FUNCTION_BLOCK Component EXTENDS FB_ComponentBase
VAR
	ComponentAlarms	 : ARRAY[1..COMPONENT_ALARM_COUNT] OF FB_TcAlarm;
	testError		 : BOOL;
	_ErrorSeverity	 : INT := 2;
	_WarningSeverity : INT;
END_VAR

VAR CONSTANT
	COMPONENT_ALARM_COUNT : UDINT := 7; //First is InitReferenceEvent
END_VAR

METHOD ChangeAlarmSeverity
CASE _WarningSeverity OF
	0:
		_ParentFaultResponseDefinitions[TcEventSeverity.Warning] := E_AlarmResponse.NoResponse;

	1:
		_ParentFaultResponseDefinitions[TcEventSeverity.Warning] := E_AlarmResponse.Abort_Immediate;

	2:
		_ParentFaultResponseDefinitions[TcEventSeverity.Warning] := E_AlarmResponse.Abort_ImmediateError;
END_CASE

CASE _ErrorSeverity OF
	0:
		_ParentFaultResponseDefinitions[TcEventSeverity.Error] := E_AlarmResponse.NoResponse;

	1:
		_ParentFaultResponseDefinitions[TcEventSeverity.Error] := E_AlarmResponse.Abort_Immediate;

	2:
		_ParentFaultResponseDefinitions[TcEventSeverity.Error] := E_AlarmResponse.Abort_ImmediateError;
END_CASE
END_METHOD

// Initializes event function blocks using this components's name
METHOD PROTECTED CreateEvents

// This method is called by Initialize() as required
F_CreateAllEventsInClass(Alarms		:= ComponentAlarms,
						 ClassSize	:= SIZEOF(TC_Events.Events_Component),
						 pInitEvent := ADR(TC_EVENTS.Events_Component.InitReferenceEvent),
						 Prefix		:= Name);

SUPER^.CreateEvents();
END_METHOD

// This method serves as the entry point for all underlying FB logic
METHOD PUBLIC CyclicLogic

// This method should be called cyclically by descendant function blocks by invoking SUPER^.CyclicLogic().  Alternatively, the contents of this method could be reimplemented entirely in which case a call to this method would not be necessary.
IF NOT _InitComplete THEN
	_InitComplete := Initialize();
	RETURN;
END_IF

//
ChangeAlarmSeverity();
SUPER^.CyclicLogic();

(*
*
*		Code must be after SUPER^.CyclicLogic();
*
*)

// Update alarm severity for this component
_CurrentAlarmSeverity := F_GetMaxSeverityRaised(Alarms := ComponentAlarms, CurrentSeverity := _CurrentAlarmSeverity);
_Error				  := _CurrentAlarmSeverity >= TcEventSeverity.Error;
END_METHOD

// Provides basic error detection and event handling for this component
METHOD PROTECTED Monitoring

//This method is called cyclically by CyclicLogic()
_Busy := FALSE;

//AlarmMonitoring
IF testError AND NOT ComponentAlarms[E_Events_Component.Error].bRaised THEN
	RaiseAlarm2Args(ComponentAlarms[E_Events_Component.Error], 'Note 1', 'Note 2');
END_IF

SUPER^.Monitoring();
END_METHOD

METHOD RaiseAlarm2Args
VAR_IN_OUT
	Alarm : FB_TcAlarm; //Alarm to be raised
END_VAR

VAR_INPUT
	String_1 : STRING; //First String Parameter (The Name of this component will be applied first automatically)
	String_2 : STRING; //Second String Parameter
END_VAR
F_RaiseAlarmWithStringParameters(Alarm	  := Alarm,
								 String_1 := Name,
								 String_2 := String_1,
								 String_3 := String_2);
END_METHOD

// Clears error flags and error IDs for this component
METHOD PUBLIC Reset : BOOL

//Typically called by the EMs SUPER^.Clearing Method
F_ClearAllEventsInClass(Alarms := ComponentAlarms);
IF SUPER^.Reset() THEN
	_Error	 := FALSE;
	_ErrorID := 0;
	Reset	 := TRUE;
END_IF
END_METHOD

END_FUNCTION_BLOCK

(* stored: Version 1.1.0.1
   POU Component: Id {b36b2c18-61ed-4d82-849b-c4ab8043897f}, SpecialFunc None
   Method ChangeAlarmSeverity: Id {a3edb0f9-f0d5-4ad0-928e-55bb25bfc45a}
   Method CreateEvents: Id {b63661ac-39bc-48a5-a0dc-7e1dceb7a9cb}
   Method CyclicLogic: Id {57f3e089-87ec-40e9-8d89-c2565e148729}
   Method Monitoring: Id {7c9b6c42-8fe1-4877-98d5-b7e6e33b37fa}
   Method RaiseAlarm2Args: Id {741dfd78-f38e-446f-bb3c-e2492225744e}
   Method Reset: Id {6737e5cc-5e58-4d89-aac0-5f2239d825cd} *)
